KUKA KRL program: art_cycle.src, art_cycle.dat

--- art_cycle.src ---
&ACCESS RVO1
&REL 54
&PARAM DISKPATH = KRC:\R1\Program\UGK
DEF art_cycle()
   DECL INT line_num

   ; Select ready work area.
   ART_PP_Select()

   ; Reset line work areas, when scheme changed.
   ART_PP_sheme_changed()

   ; Pallet filling.
   line_num = ART_line_Select()

   IF (line_num == 1) OR (line_num == 2) THEN
      ; First layer sheet.
      IF (ART_line[line_num].current_bag == 0) THEN
         move_get_sheet(1)
         move_put_sheet(line_num)
      ENDIF
      ; Product.
      ART_line_calc_next(line_num)
      move_get(line_num)
      ARTGripperGrip()
      move_put(line_num, ART_line[line_num].scheme_number)

      ARTStatProductCycle()
      ART_line_last_num = line_num
      ; Layer sheet.
      IF (ART_line[line_num].isLayerDone) THEN
         move_get_sheet(2)
         move_put_sheet(line_num)
      ENDIF
   ELSE
      art_move_center()
   ENDIF

   ; Pallet full.
   FOR line_num = 1 TO DEF_LINE_COUNT
      IF ART_line[line_num].isPalletDone THEN
         ART_PP_Full(line_num)
         ARTStatPalletCycle(line_num)
      ENDIF
   ENDFOR
END
;
; Put product on pallet.
;
DEF move_put(line_num:IN, scheme:IN)
   DECL INT line_num
   DECL INT scheme
   DECL INT wa_base

   move_pp_after(line_num)
   ART_move_center()

   wa_base = line_num + 2
   $BWDSTART=FALSE
   SWITCH wa_base
      CASE 3
         PDAT_ACT={VEL 100.000,ACC 100.000,APO_DIST 400.000,APO_MODE #CDIS,GEAR_JERK 50.0000,EXAX_IGN 0}
         FDAT_ACT={TOOL_NO 0,BASE_NO 3,IPO_FRAME #BASE,POINT2[] " ",TQ_STATE FALSE}
         BAS(#PTP_PARAMS,100)
         PTP {A1 80, A2 -72,A3 60} C_DIS
      CASE 4
         PDAT_ACT={VEL 100.000,ACC 100.000,APO_DIST 400.000,APO_MODE #CDIS,GEAR_JERK 50.0000,EXAX_IGN 0}
         FDAT_ACT={TOOL_NO 0,BASE_NO 4,IPO_FRAME #BASE,POINT2[] " ",TQ_STATE FALSE}
         BAS(#PTP_PARAMS,100)
         PTP {A1 30, A2 -110,A3 86,A6 -60} C_DIS
   ENDSWITCH
   SWITCH line_num
      CASE 1
         ;PTP
         SWITCH scheme
            CASE 1
               ;art_chah_ln1_5l(wa_base, ART_line[line_num].current_bag)
            CASE 2
               ;art_chah_ln1_10l(wa_base, ART_line[line_num].current_bag)
            DEFAULT
               ARTControlMotionCmd = #ARTMotionNone
         ENDSWITCH
      CASE 2
         ;PTP
         SWITCH scheme
            CASE 1
               ;art_chah_ln2_5l(wa_base, ART_line[line_num].current_bag)
            CASE 2
               ;art_chah_ln2_10l(wa_base, ART_line[line_num].current_bag)
            DEFAULT
               ARTControlMotionCmd = #ARTMotionNone
         ENDSWITCH
   ENDSWITCH

   ART_move_center()
END
;
; Product getting.
;
DEF move_get(line_num: IN)
   DECL INT line_num
   ;ARTForkClose()
   SWITCH line_num
      CASE 1
         ;FOLD PTP spo1 CONT Vel=100 % PDAT1 Tool[1]:calibr Base[3]:wa1;%{PE}%R 8.3.44,%MKUKATPBASIS,%CMOVE,%VPTP,%P 1:PTP, 2:spo1, 3:C_DIS, 5:100, 7:PDAT1
         $BWDSTART=FALSE
         PDAT_ACT={VEL 100.000,ACC 100.000,APO_DIST 100.000,APO_MODE #CDIS,GEAR_JERK 50.0000,EXAX_IGN 0}
         FDAT_ACT=Fspo1
         BAS(#PTP_PARAMS,100)
         PTP {A1 80, A2 -100,A3 80,A6 0} C_DIS
         ;ENDFOLD
      CASE 2
         ;FOLD PTP spo2 CONT Vel=100 % PDAT3 Tool[0] Base[2]:pick_p2;%{PE}%R 8.3.44,%MKUKATPBASIS,%CMOVE,%VPTP,%P 1:PTP, 2:spo2, 3:C_DIS, 5:100, 7:PDAT3
         $BWDSTART=FALSE
         PDAT_ACT={VEL 100.000,ACC 100.000,APO_DIST 100.000,APO_MODE #CDIS,GEAR_JERK 50.0000,EXAX_IGN 0}
         FDAT_ACT=Fspo2
         BAS(#PTP_PARAMS,100)
         PTP {A1 -90, A2 -81,A3 64,A6 -180} C_DIS
         ;ENDFOLD
   ENDSWITCH

   ART_move_pre_pp(line_num)
   ART_move_pick_point(line_num)
END
;
; Put sheet on pallet.
;
DEF move_put_sheet(line_num:IN)
   DECL INT line_num
   DECL INT wa_base

   ART_move_center()

   wa_base = line_num + 2
   $BWDSTART=FALSE
   SWITCH wa_base
      CASE 3
         PDAT_ACT={VEL 100.000,ACC 100.000,APO_DIST 400.000,APO_MODE #CDIS,GEAR_JERK 50.0000,EXAX_IGN 0}
         FDAT_ACT={TOOL_NO 0,BASE_NO 3,IPO_FRAME #BASE,POINT2[] " ",TQ_STATE FALSE}
         BAS(#PTP_PARAMS,100)
         ;PTP {A1 80, A2 -72,A3 60} C_DIS
      CASE 4
         PDAT_ACT={VEL 100.000,ACC 100.000,APO_DIST 400.000,APO_MODE #CDIS,GEAR_JERK 50.0000,EXAX_IGN 0}
         FDAT_ACT={TOOL_NO 0,BASE_NO 4,IPO_FRAME #BASE,POINT2[] " ",TQ_STATE FALSE}
         BAS(#PTP_PARAMS,100)
         ;PTP {A1 30, A2 -110,A3 86,A6 -60} C_DIS
   ENDSWITCH
   ;PTP
   ARTGripVacuumRelease()
   ;PTP
   ART_move_center()
END
;
; Sheet getting.
;
DEF move_get_sheet(stack_num:IN)
   DECL INT stack_num
   INTERRUPT DECL 21 WHEN $MEAS_PULSE[5]==FALSE DO StopMoving( )
   INTERRUPT OFF 21
   ARTStackMuteOFF(stack_num)
   $PAL_MODE = FALSE

   SWITCH stack_num
      CASE 1
         ;FOLD PTP spo1 CONT Vel=100 % PDAT1 Tool[1]:calibr Base[3]:wa1;%{PE}%R 8.3.44,%MKUKATPBASIS,%CMOVE,%VPTP,%P 1:PTP, 2:spo1, 3:C_DIS, 5:100, 7:PDAT1
         $BWDSTART=FALSE
         PDAT_ACT={VEL 100.000,ACC 100.000,APO_DIST 100.000,APO_MODE #CDIS,GEAR_JERK 50.0000,EXAX_IGN 0}
         FDAT_ACT=Fspo1
         BAS(#PTP_PARAMS,100)
         PTP {A1 80, A2 -100,A3 80,A6 0} C_DIS
         ;ENDFOLD
         ;FOLD PTP sheet1 CONT Vel=100 % PDAT4 Tool[0] Base[2]:pp2;%{PE}%R 8.3.44,%MKUKATPBASIS,%CMOVE,%VPTP,%P 1:PTP, 2:sheet1, 3:C_DIS, 5:100, 7:PDAT4
         $BWDSTART=FALSE
         PDAT_ACT=PPDAT4
         FDAT_ACT=Fsheet1
         BAS(#PTP_PARAMS,100)
         PTP {X 0,Y 0,Z 800,A 0,B 0,C 0}:Xsheet1 C_DIS
         ;ENDFOLD

         INTERRUPT ON 21
         sheets_stack_scan(stack_num)
         INTERRUPT OFF 21

         ARTGripVacuumGrip()
         ;FOLD PTP sheet1 CONT Vel=100 % PDAT4 Tool[0] Base[2]:pp2;%{PE}%R 8.3.44,%MKUKATPBASIS,%CMOVE,%VPTP,%P 1:PTP, 2:sheet1, 3:C_DIS, 5:100, 7:PDAT4
         $BWDSTART=FALSE
         PDAT_ACT=PPDAT4
         FDAT_ACT=Fsheet1
         BAS(#PTP_PARAMS,100)
         LIN {X 0,Y 0,Z 800,A 0,B 0,C 0}:Xsheet1 C_DIS C_DIS
         ;ENDFOLD
      CASE 2
         INTERRUPT DECL 21 WHEN $MEAS_PULSE[5]==FALSE DO StopMoving( )
         INTERRUPT OFF 21
         $PAL_MODE = FALSE

         ;FOLD PTP spo1 CONT Vel=100 % PDAT1 Tool[1]:calibr Base[3]:wa1;%{PE}%R 8.3.44,%MKUKATPBASIS,%CMOVE,%VPTP,%P 1:PTP, 2:spo1, 3:C_DIS, 5:100, 7:PDAT1
         $BWDSTART=FALSE
         PDAT_ACT={VEL 100.000,ACC 100.000,APO_DIST 100.000,APO_MODE #CDIS,GEAR_JERK 50.0000,EXAX_IGN 0}
         FDAT_ACT=Fspo1
         BAS(#PTP_PARAMS,100)
         PTP {A1 80, A2 -100,A3 80,A6 0} C_DIS
         ;ENDFOLD

         ;FOLD PTP sheet2 CONT Vel=100 % PDAT6 Tool[0] Base[2]:pp2;%{PE}%R 8.3.44,%MKUKATPBASIS,%CMOVE,%VPTP,%P 1:PTP, 2:sheet2, 3:C_DIS, 5:100, 7:PDAT6
         $BWDSTART=FALSE
         PDAT_ACT=PPDAT6
         FDAT_ACT=Fsheet2
         BAS(#PTP_PARAMS,100)
         PTP {X 0,Y 0,Z 800,A 0,B 0,C 0}:Xsheet2 C_DIS
         ;ENDFOLD
         INTERRUPT ON 21
         sheets_stack_scan(stack_num)
         INTERRUPT OFF 21
         ;FOLD PTP sheet2 CONT Vel=100 % PDAT6 Tool[0] Base[2]:pp2;%{PE}%R 8.3.44,%MKUKATPBASIS,%CMOVE,%VPTP,%P 1:PTP, 2:sheet2, 3:C_DIS, 5:100, 7:PDAT6
         $BWDSTART=FALSE
         PDAT_ACT=PPDAT6
         FDAT_ACT=Fsheet2
         BAS(#PTP_PARAMS,100)
         PTP {X 0,Y 0,Z 800,A 0,B 0,C 0}:Xsheet2 C_DIS
         ;ENDFOLD
   ENDSWITCH
   ARTStackMuteON(stack_num)
END
;
;
;
DEF sheets_stack_scan(stack_num: IN)
   DECL INT stack_num

   SWITCH stack_num
      CASE 1
         ARTStackLowReset(stack_num)
         ;FOLD PTP sheet1 CONT Vel=100 % PDAT4 Tool[0] Base[2]:pp2;%{PE}%R 8.3.44,%MKUKATPBASIS,%CMOVE,%VPTP,%P 1:PTP, 2:sheet1, 3:C_DIS, 5:100, 7:PDAT4
         $BWDSTART=FALSE
         PDAT_ACT=PPDAT4
         FDAT_ACT=Fsheet1
         BAS(#PTP_PARAMS,100)
         PTP {X 0,Y 0,Z 100,A 0,B 0,C 0}:Xsheet1 C_DIS
         ;ENDFOLD
         ARTStackLow(stack_num)
         ;FOLD PTP sheet1 CONT Vel=100 % PDAT4 Tool[0] Base[2]:pp2;%{PE}%R 8.3.44,%MKUKATPBASIS,%CMOVE,%VPTP,%P 1:PTP, 2:sheet1, 3:C_DIS, 5:100, 7:PDAT4
         $BWDSTART=FALSE
         PDAT_ACT=PPDAT4
         FDAT_ACT=Fsheet1
         BAS(#PTP_PARAMS,100)
         PTP Xsheet1 C_DIS
         ;ENDFOLD
      CASE 2
         ARTStackLowReset(stack_num)
         ;FOLD PTP sheet2 CONT Vel=100 % PDAT6 Tool[0] Base[2]:pp2;%{PE}%R 8.3.44,%MKUKATPBASIS,%CMOVE,%VPTP,%P 1:PTP, 2:sheet2, 3:C_DIS, 5:100, 7:PDAT6
         $BWDSTART=FALSE
         PDAT_ACT=PPDAT6
         FDAT_ACT=Fsheet2
         BAS(#PTP_PARAMS,100)
         PTP {X 0,Y 0,Z 100,A 0,B 0,C 0}:Xsheet2 C_DIS
         ;ENDFOLD
         ARTStackLow(stack_num)
         ;FOLD PTP sheet2 CONT Vel=100 % PDAT6 Tool[0] Base[2]:pp2;%{PE}%R 8.3.44,%MKUKATPBASIS,%CMOVE,%VPTP,%P 1:PTP, 2:sheet2, 3:C_DIS, 5:100, 7:PDAT6
         $BWDSTART=FALSE
         PDAT_ACT=PPDAT6
         FDAT_ACT=Fsheet2
         BAS(#PTP_PARAMS,100)
         PTP Xsheet2 C_DIS
         ;ENDFOLD
   ENDSWITCH
END
;
;
;
DEF StopMoving()
   BRAKE
   RESUME
END

--- art_cycle.dat ---
&ACCESS RVO1
&REL 54
&PARAM DISKPATH = KRC:\R1\Program\UGK
DEFDAT  art_cycle PUBLIC


; Points
DECL AXIS ASPO1={A1 80.0000,A2 -100.000,A3 80.0000,A6 0.0}
DECL AXIS ASPO2={A1 -90.0000,A2 -81.0000,A3 64.0000,A6 -180.000}
DECL AXIS Aspo_put1={A1 80.0000,A2 -72.0000,A3 60.0000} ;,A6 -28
DECL AXIS Aspo_put2={A1 30.0000,A2 -110.000,A3 86.0000,A6 -60.0000}
DECL AXIS Aspo_put4={A1 -20.0000,A2 -110.000,A3 86.0000,A6 -111.000}
DECL AXIS Aspo_put3={A1 -80.0000,A2 -72.0000,A3 60.0000}

DECL PDAT PPDAT5={VEL 100.000,ACC 100.000,APO_DIST 100.000,APO_MODE #CDIS,GEAR_JERK 50.0000,EXAX_IGN 0}
DECL LDAT LCPDAT2={VEL 2.00000,ACC 100.000,APO_DIST 100.000,APO_FAC 50.0000,AXIS_VEL 100.000,AXIS_ACC 100.000,ORI_TYP #VAR,CIRC_TYP #BASE,JERK_FAC 50.0000,GEAR_JERK 50.0000,EXAX_IGN 0}
DECL BASIS_SUGG_T LAST_BASIS={POINT1[] "sheet2                  ",POINT2[] "sheet2                  ",CP_PARAMS[] "CPDAT3                  ",PTP_PARAMS[] "PDAT6                   ",CONT[] "C_DIS                   ",CP_VEL[] "2                       ",PTP_VEL[] "100                     ",SYNC_PARAMS[] "SYNCDAT                 ",SPL_NAME[] "S0                      ",A_PARAMS[] "ADAT0                   "}
DECL E6POS XSPO1={X 998.055,Y 609.623047,Z -188.864197,A 89.8975754,B -0.248162299,C 179.934601,S 2,T 42,E1 0.0,E2 0.0,E3 0.0,E4 0.0,E5 0.0,E6 0.0}
DECL FDAT Fspo1={TOOL_NO 0,BASE_NO 1,IPO_FRAME #BASE,POINT2[] " ",TQ_STATE FALSE}
DECL PDAT PPDAT1={VEL 100.000,ACC 100.000,APO_DIST 100.000,APO_MODE #CDIS,GEAR_JERK 50.0000,EXAX_IGN 0}
DECL E6POS XPP_AFTER={X 106.804161,Y -219.755203,Z -409.195190,A 89.7331543,B 0.00309650414,C 179.891891,S 2,T 10,E1 0.0,E2 0.0,E3 0.0,E4 0.0,E5 0.0,E6 0.0}
DECL FDAT Fpp_after={TOOL_NO 0,BASE_NO 1,IPO_FRAME #BASE,POINT2[] " ",TQ_STATE FALSE}
DECL LDAT LCPDAT1={VEL 2.00000,ACC 100.000,APO_DIST 100.000,APO_FAC 50.0000,AXIS_VEL 100.000,AXIS_ACC 100.000,ORI_TYP #VAR,CIRC_TYP #BASE,JERK_FAC 50.0000,GEAR_JERK 50.0000,EXAX_IGN 0}
DECL LDAT LCPDAT3={VEL 2.00000,ACC 100.000,APO_DIST 100.000,APO_FAC 50.0000,AXIS_VEL 100.000,AXIS_ACC 100.000,ORI_TYP #VAR,CIRC_TYP #BASE,JERK_FAC 50.0000,GEAR_JERK 50.0000,EXAX_IGN 0}
DECL E6POS XSPO_PUT={X 1374.14026,Y 60.9308167,Z -150.324661,A 178.533737,B 0.108156718,C -179.999161,S 2,T 10,E1 0.0,E2 0.0,E3 0.0,E4 0.0,E5 0.0,E6 0.0}
DECL FDAT Fspo_put={TOOL_NO 0,BASE_NO 1,IPO_FRAME #BASE,POINT2[] " ",TQ_STATE FALSE}
DECL PDAT PPDAT2={VEL 100.000,ACC 100.000,APO_DIST 400.000,APO_MODE #CDIS,GEAR_JERK 50.0000,EXAX_IGN 0}
DECL E6POS XSPO2={X 598.389709,Y 220.402435,Z -185.591400,A -95.8268585,B -0.499567837,C 179.863205,S 2,T 11,E1 0.0,E2 0.0,E3 0.0,E4 0.0,E5 0.0,E6 0.0}
DECL FDAT Fspo2={TOOL_NO 0,BASE_NO 2,IPO_FRAME #BASE,POINT2[] " ",TQ_STATE FALSE}
DECL PDAT PPDAT3={VEL 100.000,ACC 100.000,APO_DIST 100.000,APO_MODE #CDIS,GEAR_JERK 50.0000,EXAX_IGN 0}
DECL E6POS XSHEET1={X -3929.83545,Y 859.430542,Z 48.9558144,A -151.150864,B 88.4548416,C 28.5093346,S 2,T 34,E1 0.0,E2 0.0,E3 0.0,E4 0.0,E5 0.0,E6 0.0}
DECL FDAT Fsheet1={TOOL_NO 0,BASE_NO 2,IPO_FRAME #BASE,POINT2[] " ",TQ_STATE FALSE}
DECL PDAT PPDAT4={VEL 100.000,ACC 100.000,APO_DIST 100.000,APO_MODE #CDIS,GEAR_JERK 50.0000,EXAX_IGN 0}
DECL E6POS XSHEET2={X -3929.83545,Y 1774.46021,Z 37.1404152,A -151.150864,B 88.4548416,C 28.5093365,S 2,T 10,E1 0.0,E2 0.0,E3 0.0,E4 0.0,E5 0.0,E6 0.0}
DECL FDAT Fsheet2={TOOL_NO 0,BASE_NO 2,IPO_FRAME #BASE,POINT2[] " ",TQ_STATE FALSE}
DECL PDAT PPDAT6={VEL 100.000,ACC 100.000,APO_DIST 100.000,APO_MODE #CDIS,GEAR_JERK 50.0000,EXAX_IGN 0}
ENDDAT
